// Mitsubishi GX Works2 project: servo6   PLC: Q03UDV

PROGRAM SERVO
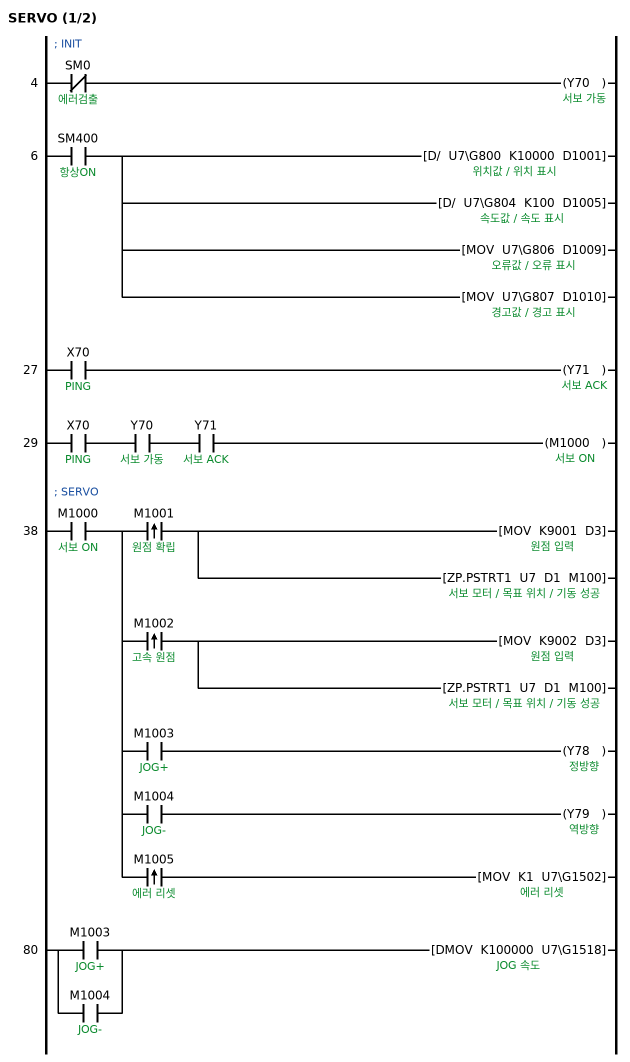
; INIT
4     LDI     SM0  ; 에러검출
      OUT     Y70  ; 서보 가동
6     LD      SM400  ; 항상ON
      D/      U7\G800 K10000 D1001  ; 위치값 / 위치 표시
      D/      U7\G804 K100 D1005  ; 속도값 / 속도 표시
      MOV     U7\G806 D1009  ; 오류값 / 오류 표시
      MOV     U7\G807 D1010  ; 경고값 / 경고 표시
27    LD      X70  ; PING
      OUT     Y71  ; 서보 ACK
29    LD      X70  ; PING
      AND     Y70  ; 서보 가동
      AND     Y71  ; 서보 ACK
      OUT     M1000  ; 서보 ON
; SERVO
38    LD      M1000  ; 서보 ON
      MPS
      ANDP    M1001  ; 원점 확립
      MOV     K9001 D3  ; 원점 입력
      ZP.PSTRT1 U7 D1 M100  ; 서보 모터 / 목표 위치 / 기동 성공
      MRD
      ANDP    M1002  ; 고속 원점
      MOV     K9002 D3
      ZP.PSTRT1 U7 D1 M100
      MRD
      AND     M1003  ; JOG+
      OUT     Y78  ; 정방향
      MRD
      AND     M1004  ; JOG-
      OUT     Y79  ; 역방향
      MPP
      ANDP    M1005  ; 에러 리셋
      MOV     K1 U7\G1502  ; 에러 리셋
80    LD      M1003  ; JOG+
      OR      M1004  ; JOG-
      DMOV    K100000 U7\G1518  ; JOG 속도
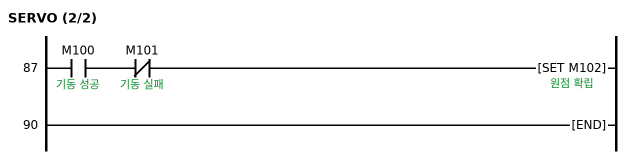
87    LD      M100  ; 기동 성공
      ANI     M101  ; 기동 실패
      SET     M102  ; 원점 확립
90    END
END_PROGRAM

PROGRAM MAIN
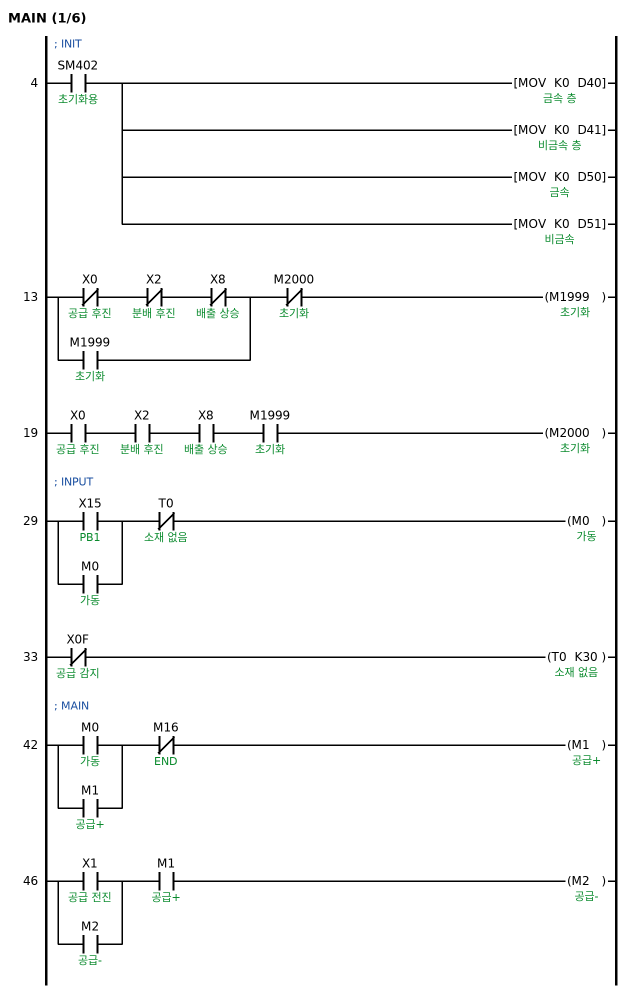
; INIT
4     LD      SM402  ; 초기화용
      MOV     K0 D40  ; 금속 층
      MOV     K0 D41  ; 비금속 층
      MOV     K0 D50  ; 금속
      MOV     K0 D51  ; 비금속
13    LDI     X0  ; 공급 후진
      ANI     X2  ; 분배 후진
      ANI     X8  ; 배출 상승
      OR      M1999  ; 초기화
      ANI     M2000  ; 초기화
      OUT     M1999  ; 초기화
19    LD      X0  ; 공급 후진
      AND     X2  ; 분배 후진
      AND     X8  ; 배출 상승
      AND     M1999  ; 초기화
      OUT     M2000  ; 초기화
; INPUT
29    LD      X15  ; PB1
      OR      M0  ; 가동
      ANI     T0  ; 소재 없음
      OUT     M0  ; 가동
33    LDI     X0F  ; 공급 감지
      OUT     T0 K30  ; 소재 없음
; MAIN
42    LD      M0  ; 가동
      OR      M1  ; 공급+
      ANI     M16  ; END
      OUT     M1  ; 공급+
46    LD      X1  ; 공급 전진
      OR      M2  ; 공급-
      AND     M1  ; 공급+
      OUT     M2  ; 공급-
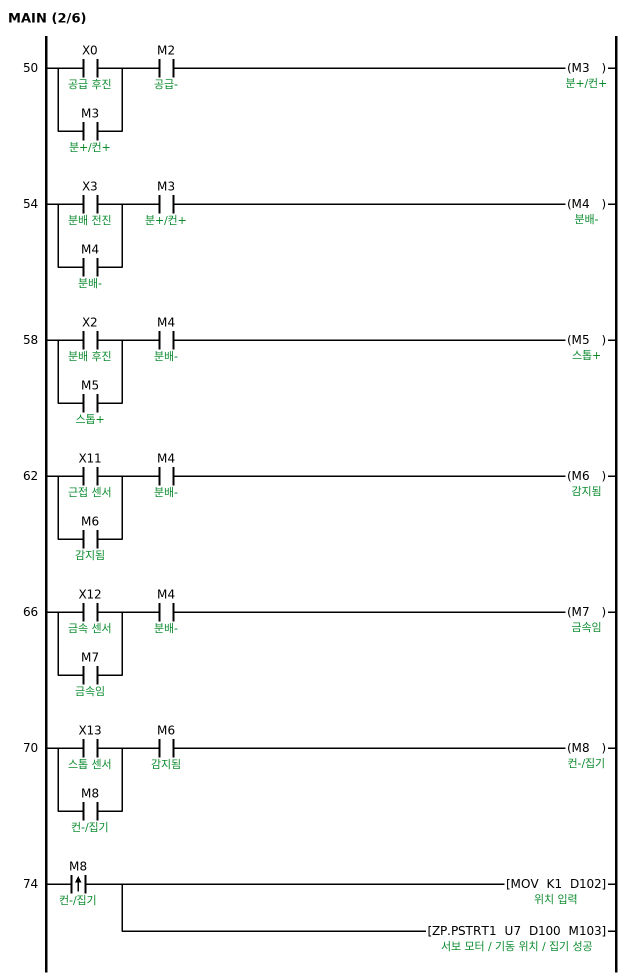
50    LD      X0  ; 공급 후진
      OR      M3  ; 분+/컨+
      AND     M2  ; 공급-
      OUT     M3  ; 분+/컨+
54    LD      X3  ; 분배 전진
      OR      M4  ; 분배-
      AND     M3  ; 분+/컨+
      OUT     M4  ; 분배-
58    LD      X2  ; 분배 후진
      OR      M5  ; 스톱+
      AND     M4  ; 분배-
      OUT     M5  ; 스톱+
62    LD      X11  ; 근접 센서
      OR      M6  ; 감지됨
      AND     M4  ; 분배-
      OUT     M6  ; 감지됨
66    LD      X12  ; 금속 센서
      OR      M7  ; 금속임
      AND     M4  ; 분배-
      OUT     M7  ; 금속임
70    LD      X13  ; 스톱 센서
      OR      M8  ; 컨-/집기
      AND     M6  ; 감지됨
      OUT     M8  ; 컨-/집기
74    LDP     M8  ; 컨-/집기
      MOV     K1 D102  ; 위치 입력
      ZP.PSTRT1 U7 D100 M103  ; 서보 모터 / 기동 위치 / 집기 성공
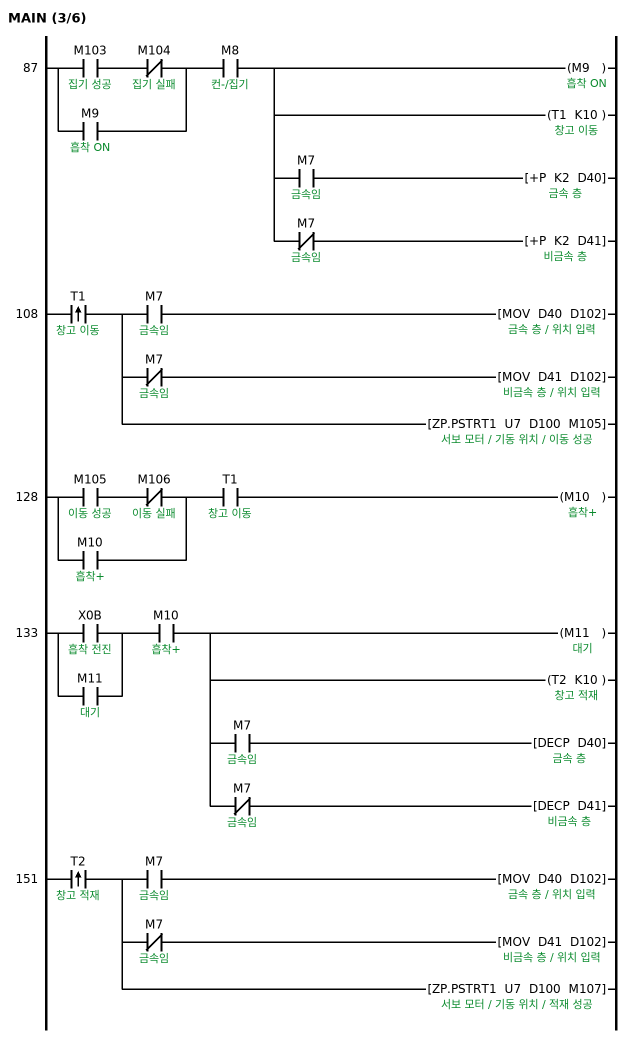
87    LD      M103  ; 집기 성공
      ANI     M104  ; 집기 실패
      OR      M9  ; 흡착 ON
      AND     M8  ; 컨-/집기
      OUT     M9  ; 흡착 ON
      OUT     T1 K10  ; 창고 이동
      MPS
      AND     M7  ; 금속임
      +P      K2 D40
      MPP
      ANI     M7  ; 금속임
      +P      K2 D41
108   LDP     T1  ; 창고 이동
      MPS
      AND     M7  ; 금속임
      MOV     D40 D102
      MRD
      ANI     M7  ; 금속임
      MOV     D41 D102
      MPP
      ZP.PSTRT1 U7 D100 M105  ; 이동 성공
128   LD      M105  ; 이동 성공
      ANI     M106  ; 이동 실패
      OR      M10  ; 흡착+
      AND     T1  ; 창고 이동
      OUT     M10  ; 흡착+
133   LD      X0B  ; 흡착 전진
      OR      M11  ; 대기
      AND     M10  ; 흡착+
      OUT     M11  ; 대기
      OUT     T2 K10  ; 창고 적재
      MPS
      AND     M7  ; 금속임
      DECP    D40
      MPP
      ANI     M7  ; 금속임
      DECP    D41
151   LDP     T2  ; 창고 적재
      MPS
      AND     M7  ; 금속임
      MOV     D40 D102
      MRD
      ANI     M7  ; 금속임
      MOV     D41 D102
      MPP
      ZP.PSTRT1 U7 D100 M107  ; 적재 성공
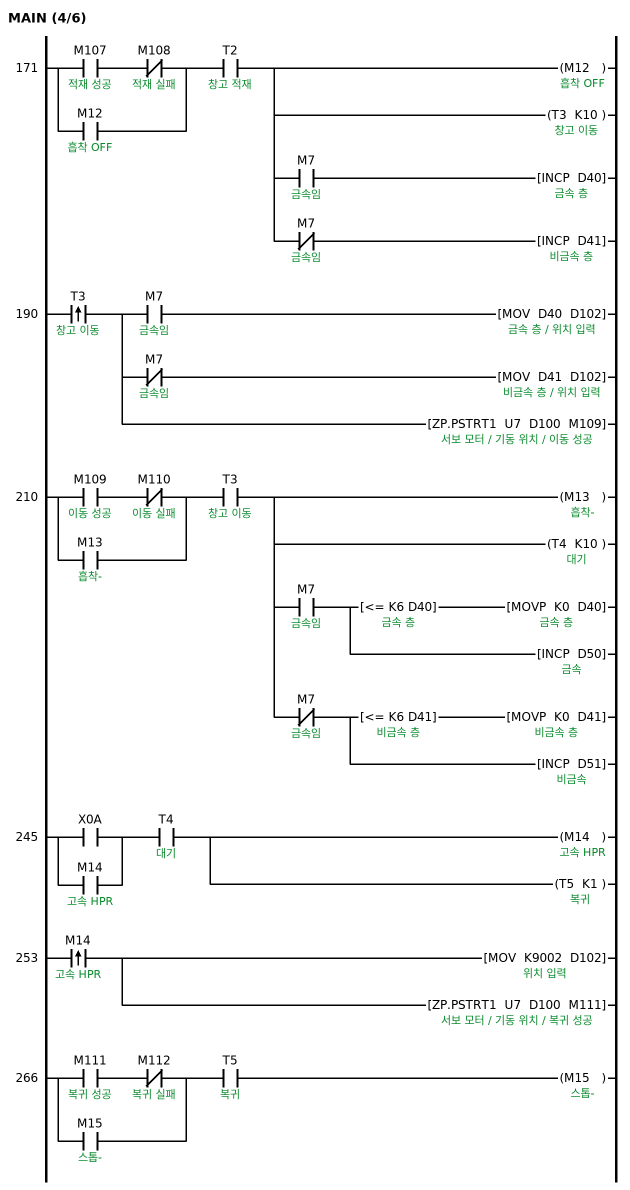
171   LD      M107  ; 적재 성공
      ANI     M108  ; 적재 실패
      OR      M12  ; 흡착 OFF
      AND     T2  ; 창고 적재
      OUT     M12  ; 흡착 OFF
      OUT     T3 K10  ; 창고 이동
      MPS
      AND     M7  ; 금속임
      INCP    D40
      MPP
      ANI     M7  ; 금속임
      INCP    D41
190   LDP     T3  ; 창고 이동
      MPS
      AND     M7  ; 금속임
      MOV     D40 D102
      MRD
      ANI     M7  ; 금속임
      MOV     D41 D102
      MPP
      ZP.PSTRT1 U7 D100 M109  ; 이동 성공
210   LD      M109  ; 이동 성공
      ANI     M110  ; 이동 실패
      OR      M13  ; 흡착-
      AND     T3  ; 창고 이동
      OUT     M13  ; 흡착-
      OUT     T4 K10  ; 대기
      MPS
      AND     M7  ; 금속임
      MPS
      AND<=   K6 D40  ; 금속 층
      MOVP    K0 D40
      MPP
      INCP    D50
      MPP
      ANI     M7  ; 금속임
      MPS
      AND<=   K6 D41  ; 비금속 층
      MOVP    K0 D41
      MPP
      INCP    D51
245   LD      X0A
      OR      M14  ; 고속 HPR
      AND     T4  ; 대기
      OUT     M14  ; 고속 HPR
      OUT     T5 K1  ; 복귀
253   LDP     M14  ; 고속 HPR
      MOV     K9002 D102
      ZP.PSTRT1 U7 D100 M111  ; 복귀 성공
266   LD      M111  ; 복귀 성공
      ANI     M112  ; 복귀 실패
      OR      M15  ; 스톱-
      AND     T5  ; 복귀
      OUT     M15  ; 스톱-
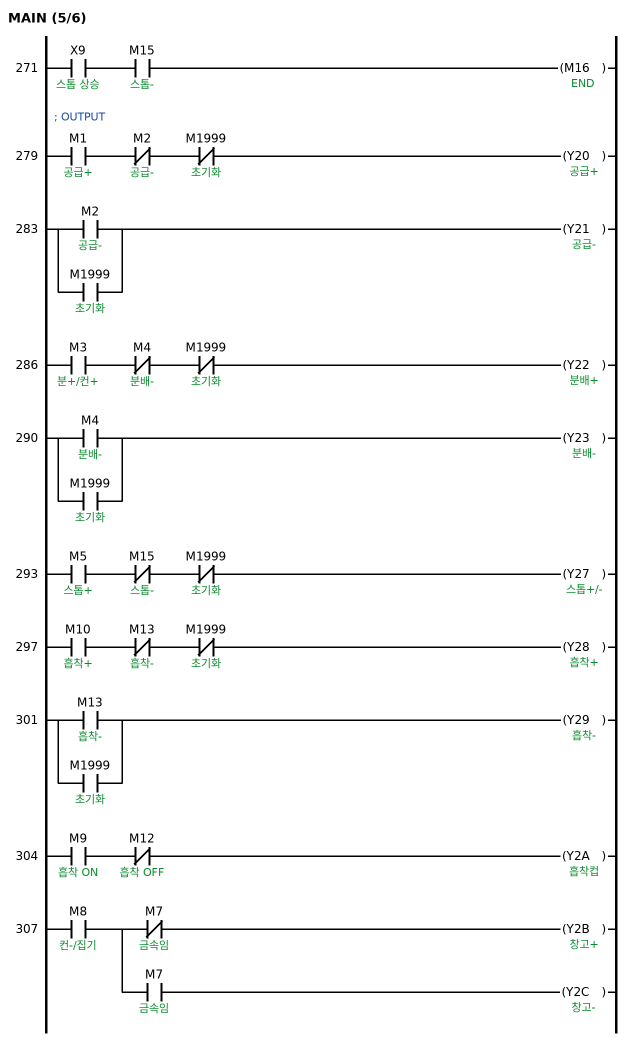
271   LD      X9  ; 스톱 상승
      AND     M15  ; 스톱-
      OUT     M16  ; END
; OUTPUT
279   LD      M1  ; 공급+
      ANI     M2  ; 공급-
      ANI     M1999  ; 초기화
      OUT     Y20  ; 공급+
283   LD      M2  ; 공급-
      OR      M1999  ; 초기화
      OUT     Y21  ; 공급-
286   LD      M3  ; 분+/컨+
      ANI     M4  ; 분배-
      ANI     M1999  ; 초기화
      OUT     Y22  ; 분배+
290   LD      M4  ; 분배-
      OR      M1999  ; 초기화
      OUT     Y23  ; 분배-
293   LD      M5  ; 스톱+
      ANI     M15  ; 스톱-
      ANI     M1999  ; 초기화
      OUT     Y27  ; 스톱+/-
297   LD      M10  ; 흡착+
      ANI     M13  ; 흡착-
      ANI     M1999  ; 초기화
      OUT     Y28  ; 흡착+
301   LD      M13  ; 흡착-
      OR      M1999  ; 초기화
      OUT     Y29  ; 흡착-
304   LD      M9  ; 흡착 ON
      ANI     M12  ; 흡착 OFF
      OUT     Y2A  ; 흡착컵
307   LD      M8  ; 컨-/집기
      MPS
      ANI     M7  ; 금속임
      OUT     Y2B  ; 창고+
      MPP
      AND     M7  ; 금속임
      OUT     Y2C  ; 창고-
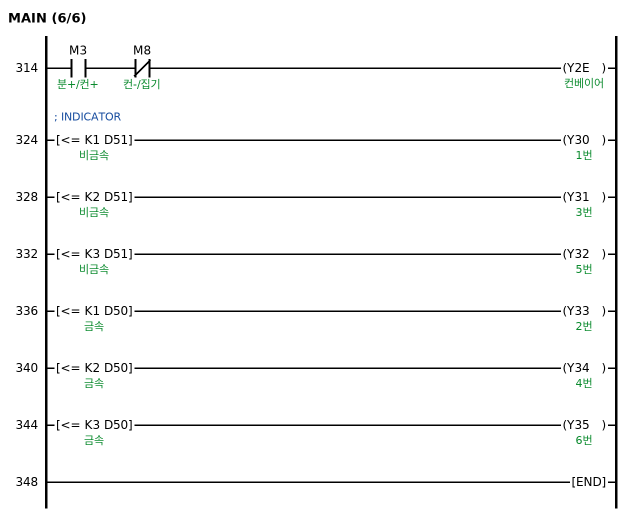
314   LD      M3  ; 분+/컨+
      ANI     M8  ; 컨-/집기
      OUT     Y2E  ; 컨베이어
; INDICATOR
324   LD<=    K1 D51  ; 비금속
      OUT     Y30  ; 1번
328   LD<=    K2 D51  ; 비금속
      OUT     Y31  ; 3번
332   LD<=    K3 D51  ; 비금속
      OUT     Y32  ; 5번
336   LD<=    K1 D50  ; 금속
      OUT     Y33  ; 2번
340   LD<=    K2 D50  ; 금속
      OUT     Y34  ; 4번
344   LD<=    K3 D50  ; 금속
      OUT     Y35  ; 6번
348   END
END_PROGRAM

// device comments not shown above
D30  ; 층 수
M200  ; 기동 성공
